SUBAPPLICATION Uebung_171b_ASR (* Exercise for ASR_AX_SR, ueber AE-Adapter statt rohe Events (ASR_2AE_TO_SR statt ASR_2EVENTS_TO_SR) *)
  (* Standard: 61499-2; Description: Copyright (c) 2026 Meisterschulen am Ostbahnhof This program and the accompanying materials are made available under the terms of the Eclipse Public License 2.0 which is available at https://www.eclipse.org/legal/epl-2.0/ SPDX-License-Identifier: EPL-2.0 *)
  (* Version 1.0, 2026-09-07, Franz Höpfinger, Meisterschulen am Ostbahnhof, initial API and implementation and/or initial documentation *)
  PACKAGE Uebungen;
  IMPORT logiBUS::io::DI::logiBUS_DI::Input_I1;
  IMPORT logiBUS::io::DI::logiBUS_DI::Input_I2;
  IMPORT logiBUS::io::DI::logiBUS_DI_Events::BUTTON_SINGLE_CLICK;
  IMPORT logiBUS::io::DQ::logiBUS_DO::Output_Q1;
  (* Documentation:
  SET/RESET über AE-Adapter statt rohe Events
   Dieselbe Funktion wie Uebung_171_ASR (I1 = SET-Klick, I2 = RESET-Klick, Latch via ASR_AX_SR), aber der Umweg über ASR_2AE_TO_SR statt ASR_2EVENTS_TO_SR zeigt, WARUM es den AE-Adapter-Weg überhaupt gibt.
   Funktionsbeschreibung
    - ASR_2EVENTS_TO_SR (in Uebung_171_ASR) hat rohe EventInputs - jede beliebige Event-Quelle passt direkt, ohne Typ-Zwang, aber auch ohne dass sich das Signal wie ein Adapter weiterverarbeiten lässt.
   - ASR_2AE_TO_SR hat stattdessen SET_IN/RESET_IN als AE-Adapter-Sockets - die Quelle muss selbst einen AE-Plug liefern. AE_EVENT_TO_E baut die Brücke: rohes Klick-Event (logiBUS_IE.IND) hinein, getypter AE-Plug heraus.
   - Der Gewinn: ein AE-Plug ist ein normaler Adapter wie AX/ASR/ASRT - er lässt sich mit AE_SPLIT_2 vervielfältigen oder mit einem künftigen AE_MERGE_2 zusammenführen, genau wie es Uebung_231_AX für ASR zeigt. Ein rohes Event kann das nicht - es ist nur über EventConnections verdrahtbar, nicht als eigenständiges, weiterreichbares Adapter-Signal.
    Arbeitsauftrag
   Testen Sie identisch zu Uebung_171_ASR: I1 klicken → Q1 EIN, I2 klicken → Q1 AUS. Vergleichen Sie im Editor beide SubApps - gleiches Verhalten, aber Uebung_171b_ASR hat zwischen Taster und Latch zwei zusätzliche AE_EVENT_TO_E-Bausteine.
  *)
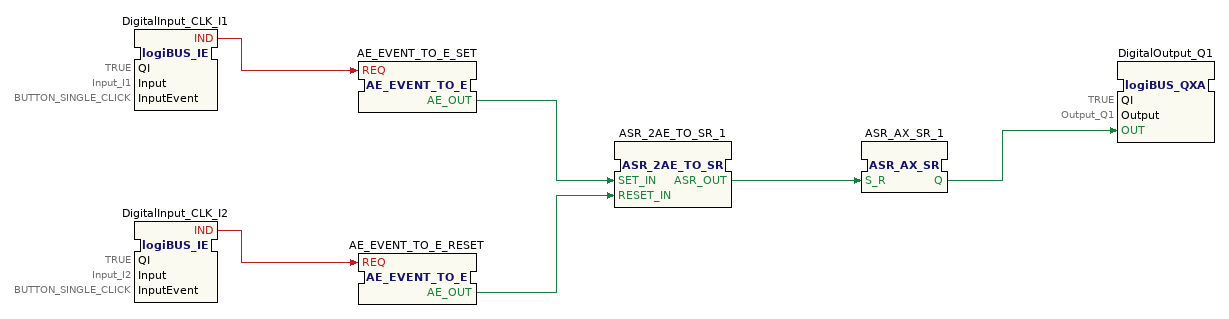
  (* Vergleich zu Uebung_171_ASR: dort ASR_2EVENTS_TO_SR mit rohen EventInputs (jede beliebige Quelle passt, ohne Typ). Hier ASR_2AE_TO_SR mit AE-Adapter-Sockets: die Quelle muss selbst einen AE-Plug liefern - AE_EVENT_TO_E baut die Bruecke vom rohen Klick-Event zum typisierten AE. Vorteil: AE-Plugs lassen sich wie jeder Adapter mit AE_SPLIT_2/AE_MERGE_2 weiterverarbeiten, ein rohes Event nicht. *)
  FBS
    ASR_AX_SR_1 : adapter::events::unidirectional::ASR_AX_SR;
    ASR_2AE_TO_SR_1 : adapter::conversion::unidirectional::ASR_2AE_TO_SR;
    AE_EVENT_TO_E_SET : adapter::conversion::unidirectional::AE_EVENT_TO_E;
    AE_EVENT_TO_E_RESET : adapter::conversion::unidirectional::AE_EVENT_TO_E;
    DigitalInput_CLK_I1 : logiBUS::io::DI::logiBUS_IE(QI := TRUE, Input := Input_I1, InputEvent := BUTTON_SINGLE_CLICK);
    DigitalOutput_Q1 : logiBUS::io::DQ::logiBUS_QXA(QI := TRUE, Output := Output_Q1);
    DigitalInput_CLK_I2 : logiBUS::io::DI::logiBUS_IE(QI := TRUE, Input := Input_I2, InputEvent := BUTTON_SINGLE_CLICK);
  END_FBS
  EVENT_CONNECTIONS
    DigitalInput_CLK_I1.IND TO AE_EVENT_TO_E_SET.REQ;
    DigitalInput_CLK_I2.IND TO AE_EVENT_TO_E_RESET.REQ;
  END_CONNECTIONS
  ADAPTER_CONNECTIONS
    AE_EVENT_TO_E_SET.AE_OUT TO ASR_2AE_TO_SR_1.SET_IN;
    AE_EVENT_TO_E_RESET.AE_OUT TO ASR_2AE_TO_SR_1.RESET_IN;
    ASR_2AE_TO_SR_1.ASR_OUT TO ASR_AX_SR_1.S_R;
    ASR_AX_SR_1.Q TO DigitalOutput_Q1.OUT;
  END_CONNECTIONS
END_SUBAPPLICATION
